PROGRAM MAIN
VAR
    level : WORD := 0;
    pump : BOOL := FALSE;
    low : BOOL;
    high : BOOL;
    low_3 : INT := 0;
    high_3 : INT := 3;
END_VAR

level := GVL.mb_Output_Registers[0];

low := level <=  low_3;
high := level >= high_3;
pump := NOT(low) AND (high OR pump);

GVL.mb_Input_Coils[0] := pump;

END_PROGRAM

(* stored: Version 1.1.0.1
   POU MAIN: Id {e13b48cb-c3c0-48f4-8553-416c703237f6}, SpecialFunc None *)
